INTERFACE I_ParameterUpdatedEvent EXTENDS I_Event

PROPERTY PUBLIC TargetParameter : I_Parameter
GET
END_GET
END_PROPERTY

END_INTERFACE

(* stored: Version 1.1.0.1, ProductVersion 3.1.4024.13
   Itf I_ParameterUpdatedEvent: Id {92d908a0-55da-050d-1ac0-428c751ab08e}
   Property TargetParameter: Id {6a3e5594-04ae-06c2-2604-265f8ed5aa0b}
   Get Get: Id {d2c8240a-f137-0706-0039-2b4da5b0831f} *)
